FUNCTION_BLOCK EL2014
VAR
	{attribute addProperty Name "WcState"}
	_wcState : WcStateInputToggle;
	{attribute addProperty Name "Info data"}
	_infoData : InfoDataAds;
	_io : EL2014_Data;
END_VAR

PROPERTY IO : REFERENCE TO EL2014_Data
GET
IO REF= _io;
END_GET
END_PROPERTY

PROPERTY WcState : REFERENCE TO WcStateInputToggle
GET
WcState REF= _wcState;
END_GET
END_PROPERTY

END_FUNCTION_BLOCK

(* stored: Version 1.1.0.1, ProductVersion 3.1.4024.9
   POU EL2014: Id {004e72ac-9486-0f99-2456-888dea05c566}, SpecialFunc None
   Property IO: Id {36f115ba-c929-0934-203a-89a93c903863}
   Get Get: Id {5f03d0e3-6396-00d8-384b-0dcbbdb07987}
   Property WcState: Id {45e0171b-0e5f-0fc4-0c9f-2682f002d393}
   Get Get: Id {c86f7e9a-2e27-0f3a-075a-8eb5b4e3e1cf} *)
